TYPE ST_HMI_OtherParamsRow :
STRUCT
	Parameter : STRING(32);
    Value     : REAL;
    Units     : STRING(8);
END_STRUCT
END_TYPE

(* stored: Version 1.1.0.1, ProductVersion 3.1.4024.12
   DUT ST_HMI_OtherParamsRow: Id {1189c503-1f71-492b-9ea8-93fe9ab9b91a} *)
